TYPE EtcMasterBase_62654B43 :
STRUCT
END_STRUCT
END_TYPE

(* stored: Version 1.2.0.0, ProductVersion 3.1.4024.9
   DUT EtcMasterBase_62654B43: Id {ff9912cc-8a88-4dee-a2ed-f3f09af6852e} *)
